// TIA Portal V19 export
TYPE "A0301_Mach_Ribaltatore_Par"
   STRUCT
      SemiAut_Vel { S7_SetPoint := 'True'} : LReal;
      Aut_Vel : LReal;
      Aut_Acc { S7_SetPoint := 'True'} : LReal;
      Aut_Dec { S7_SetPoint := 'True'} : LReal;
      Pos_0 { S7_SetPoint := 'True'} : LReal;   // Posizione di attesa sotto conveyor
      Pos_1 { S7_SetPoint := 'True'} : LReal;   // Posizione Beam sollevato e attesa su L
      Pos_2 { S7_SetPoint := 'True'} : LReal;   // Posizione Beam pronto per capovolgimento
      Pos_3 { S7_SetPoint := 'True'} : LReal;   // Posizione Beam capovolto su P2
   END_STRUCT;
END_TYPE
